INTERFACE IPistonHorizontal

METHOD MoveLeft : TcoCore.ITcoTaskStatus
END_METHOD

METHOD MoveRight : TcoCore.ITcoTaskStatus
END_METHOD

END_INTERFACE

(* stored: Version 1.1.0.1, ProductVersion 3.1.4024.6
   Itf IPistonHorizontal: Id {63be3ff7-8a36-44e1-91e4-a7ee8529c39b}
   Folder Horizontal: Id {171da708-495f-4bd2-8ff7-065f165a7d2a}
   Method MoveLeft: Id {a45eb76f-ccd1-4a1d-b916-c7d83ebc818e}
   Method MoveRight: Id {3c2e2fdb-0750-4e7d-b873-31649b547b12} *)
